RoboDK station: AQIS.rdk

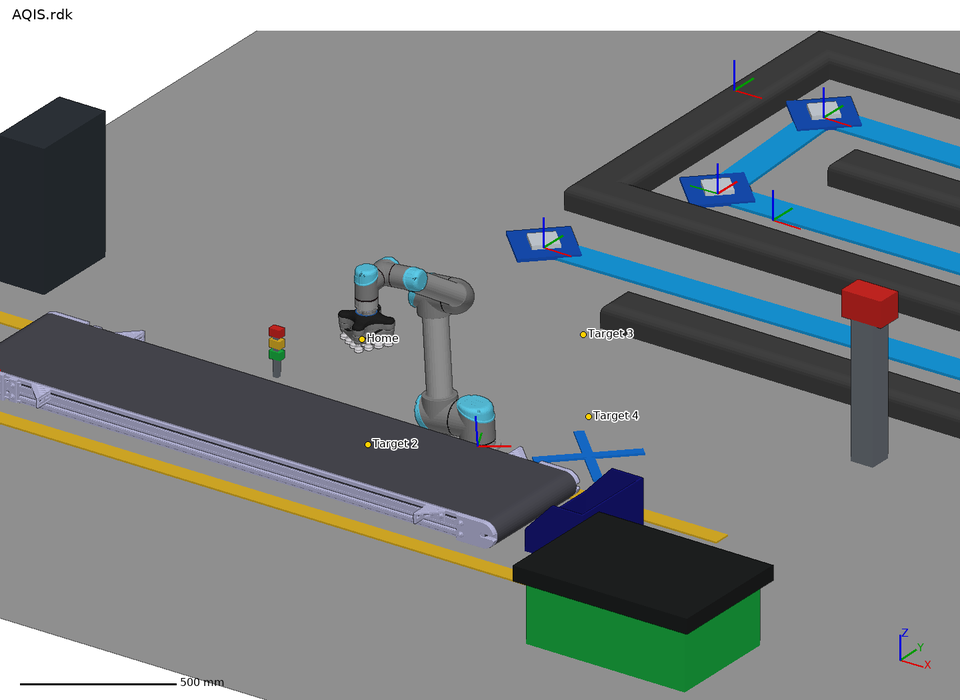
[picture v0: the station drawn from its stored meshes, robots at their saved joint values, targets as dots, program paths as lines]
Station 로봇팔 이동 (saved by RoboDK 5.7.4). Poses are relative to the parent item; angles as X-Y-Z fixed-axis rotations.
Station parameters (name, value as stored): LOAD_READY, 1, RED_DETECTED, 1, AGV_DONE, 1, CONVEYOR_DONE, 1
  - frame MainFrame at (0, 0, 0) mm
    - target Home (Cartesian target) at (651.26, -3006.26, 497.49) mm, rotated rx -179.45 ry 0.15 rz -30.37 deg; joints [-119.255, -87.831, -60.137, -122.512, 86.049, -150.839] of UR5
    - target Target 2 (Cartesian target) at (648.88, -2966.89, 106.48) mm, rotated rx -178.43 ry 0.42 rz -30.32 deg; joints [-119.274, -83.377, -123.993, -64.137, 86.304, -150.836] of UR5
    - target Target 3 (Cartesian target) at (1212.52, -2572.15, 497.3) mm, rotated rx -179.45 ry 0.15 rz -30.37 deg; joints [-13.799, -91.747, -62.441, -119.492, 91.513, -45.448] of UR5
    - target Target 4 (Cartesian target) at (1158.42, -2465.93, 148.85) mm, rotated rx -179.45 ry 0.15 rz -30.37 deg; joints [3.481, -82.996, -122.873, -67.196, 92.538, -28.188] of UR5
    - object path at (2090, -1100, 0) mm, size 3150 x 1417.4 x 86 mm, geometry from path.step
    - object path2 at (1760, -180, 0) mm, rotated rx 0 ry 0 rz 180 deg, size 3150 x 1417.4 x 86 mm, geometry from path.step
    - frame UR5 Base at (820, -2600, 0) mm, rotated rx -1.94 ry -3.6 rz 28.07 deg
      - robot UR5: 6 axes
          modified DH rows (alpha deg, a mm, theta deg, d mm): 0, 0, 0, 89.2; 90, 0, 180, 0; 0, 425, 0, 0; 0, 392, 0, 109.3; -90, 0, 0, 94.75; 90, 0, 180, 82.5
          joint limits [-360, -360, -360, -360, -360, -360] to [360, 360, 360, 360, 360, 360]; home [0, -90, -90, 0, 90, 0]; saved at [-114.958, -89.114, -59.218, -122.443, 86.096, -146.532]
        - tool OnRobot VG10 Vacuum Gripper, TCP at (-36.63, 0, 130.9) mm, size 145.4 x 145.4 x 118.3 mm
    - object Floor at (3000, -3000, 0) mm, size 3000 x 3000 x 0 mm, geometry from Floor (1).sld
    - object Floor at (0, -3000, 0) mm, size 3000 x 3000 x 0 mm, geometry from Floor (1).sld
    - object Floor at (0, 0, 0) mm, size 3000 x 3000 x 0 mm, geometry from Floor (1).sld
    - object Bin Red at (3820, 150, 0) mm, rotated rx 0 ry 0 rz -180 deg, size 225 x 337.5 x 191.2 mm, geometry from Bin-Red.sld
    - object Floor at (3000, 0, 0) mm, size 3000 x 3000 x 0 mm, geometry from Floor (1).sld
    - object Bin Blue at (1380, -2800, 0) mm, rotated rx 0 ry 0 rz -180 deg, size 225 x 337.5 x 191.2 mm, geometry from Bin-Blue.sld
    - frame Conveyor Belt (2m) Base at (-740, -3190, 100) mm
      - robot Conveyor Belt (2m): 1 axes
          modified DH rows (alpha deg, a mm, theta deg, d mm): 0, 0, 0, 0 linear
          base shift (0, 0, 0) mm, rotated rx 0 ry 90 rz 0 deg
          joint limits [-500000] to [500000]; home [0]; saved at [0]
    - frame turtlebot Base at (3580, 0, 20) mm
      - object turtlebot3_waffle at (0, 0, 0) mm, size 280.7 x 305.1 x 138.1 mm, geometry from turtlebot3_waffle (1).step
      - object Red at (48.75, 24.69, 122.77) mm, rotated rx -1.02 ry 0.28 rz -130.77 deg, size 139.8 x 166.4 x 15 mm, geometry from canlid_abnormal.step
    - frame nav1 at (160, -1290, 0) mm
    - frame nav2 at (3450, -1240, 0) mm, rotated rx 0 ry 0 rz 90 deg
    - frame nav3 at (3450, -610, 0) mm, rotated rx 0 ry 0 rz 180 deg
    - frame nav4 at (390, -650, 0) mm, rotated rx 0 ry 0 rz 90 deg
    - frame nav5 at (350, 0, 0) mm
    - frame nav6 at (3580, 0, 0) mm
    - object Blue at (1463.1, -2990, -1.25) mm, size 138.1 x 165.7 x 15 mm, geometry from canlid_normal.step
    - object Green at (1465.6, -2990, -1.25) mm, size 138.1 x 165.7 x 15 mm, geometry from canlid_normal.step
    - object Yellow at (1470.6, -2990, -1.25) mm, size 138.1 x 165.7 x 15 mm, geometry from canlid_normal.step
  - Python program Pickplace (listed below)
  - Python program Turtlebot (listed below)
  - Python program Conv (listed below)
  - Python program Main (listed below)
  - object VIS_Conveyor_Zone_Line_Left at (370, -3310, 2) mm, size 3000 x 65 x 9 mm, geometry from VIS_Conveyor_Zone_Line_Left.stl
  - object VIS_Conveyor_Zone_Line_Right at (350, -2710, 2) mm, size 3000 x 65 x 9 mm, geometry from VIS_Conveyor_Zone_Line_Right.stl
  - object VIS_AGV_Route_Line_01 at (1805, -1265, 6) mm, rotated rx 0 ry 0 rz 0.87 deg, size 3290.4 x 115 x 10 mm, geometry from VIS_AGV_Route_Line_01.stl
  - object VIS_AGV_Route_Line_02 at (3450, -925, 6) mm, rotated rx 0 ry 0 rz 90 deg, size 630 x 115 x 10 mm, geometry from VIS_AGV_Route_Line_02.stl
  - object VIS_AGV_Route_Line_03 at (1920, -630, 6) mm, rotated rx 0 ry 0 rz -179.25 deg, size 3060.3 x 115 x 10 mm, geometry from VIS_AGV_Route_Line_03.stl
  - object VIS_AGV_Route_Line_04 at (370, -325, 6) mm, rotated rx 0 ry 0 rz 93.52 deg, size 651.2 x 115 x 10 mm, geometry from VIS_AGV_Route_Line_04.stl
  - object VIS_AGV_Route_Line_05 at (1965, 0, 6) mm, size 3230 x 115 x 10 mm, geometry from VIS_AGV_Route_Line_05.stl
  - object VIS_AGV_Waypoint_01 at (160, -1290, 12) mm, rotated rx 0 ry 0 rz 45 deg, size 210 x 210 x 12 mm, geometry from VIS_AGV_Waypoint_01.stl
  - object VIS_AGV_Waypoint_Core_01 at (160, -1290, 24) mm, rotated rx 0 ry 0 rz 45 deg, size 95 x 95 x 18 mm, geometry from VIS_AGV_Waypoint_Core_01.stl
  - object VIS_AGV_Waypoint_02 at (3450, -1240, 12) mm, rotated rx 0 ry 0 rz 45 deg, size 210 x 210 x 12 mm, geometry from VIS_AGV_Waypoint_02.stl
  - object VIS_AGV_Waypoint_Core_02 at (3450, -1240, 24) mm, rotated rx 0 ry 0 rz 45 deg, size 95 x 95 x 18 mm, geometry from VIS_AGV_Waypoint_Core_02.stl
  - object VIS_AGV_Waypoint_03 at (3450, -610, 12) mm, rotated rx 0 ry 0 rz 45 deg, size 210 x 210 x 12 mm, geometry from VIS_AGV_Waypoint_03.stl
  - object VIS_AGV_Waypoint_Core_03 at (3450, -610, 24) mm, rotated rx 0 ry 0 rz 45 deg, size 95 x 95 x 18 mm, geometry from VIS_AGV_Waypoint_Core_03.stl
  - object VIS_AGV_Waypoint_04 at (390, -650, 12) mm, rotated rx 0 ry 0 rz 45 deg, size 210 x 210 x 12 mm, geometry from VIS_AGV_Waypoint_04.stl
  - object VIS_AGV_Waypoint_Core_04 at (390, -650, 24) mm, rotated rx 0 ry 0 rz 45 deg, size 95 x 95 x 18 mm, geometry from VIS_AGV_Waypoint_Core_04.stl
  - object VIS_AGV_Waypoint_05 at (350, 0, 12) mm, rotated rx 0 ry 0 rz 45 deg, size 210 x 210 x 12 mm, geometry from VIS_AGV_Waypoint_05.stl
  - object VIS_AGV_Waypoint_Core_05 at (350, 0, 24) mm, rotated rx 0 ry 0 rz 45 deg, size 95 x 95 x 18 mm, geometry from VIS_AGV_Waypoint_Core_05.stl
  - object VIS_AGV_Waypoint_06 at (3580, 0, 12) mm, rotated rx 0 ry 0 rz 45 deg, size 210 x 210 x 12 mm, geometry from VIS_AGV_Waypoint_06.stl
  - object VIS_AGV_Waypoint_Core_06 at (3580, 0, 24) mm, rotated rx 0 ry 0 rz 45 deg, size 95 x 95 x 18 mm, geometry from VIS_AGV_Waypoint_Core_06.stl
  - object VIS_AGV_Pickup_Pad_Target4 at (1158.4, -2465.9, 7) mm, rotated rx 0 ry 0 rz -45 deg, size 360 x 34 x 8 mm, geometry from VIS_AGV_Pickup_Pad_Target4.stl
  - object VIS_AGV_Pickup_Pad_Target4_Cross at (1158.4, -2465.9, 8) mm, rotated rx 0 ry 0 rz -45 deg, size 34 x 360 x 8 mm, geometry from VIS_AGV_Pickup_Pad_Target4_Cross.stl
  - object VIS_AGV_Dock_Pad_Nav6 at (3580, 0, 7) mm, size 420 x 42 x 8 mm, geometry from VIS_AGV_Dock_Pad_Nav6.stl
  - object VIS_AGV_Dock_Pad_Nav6_Cross at (3580, 0, 8) mm, size 42 x 420 x 8 mm, geometry from VIS_AGV_Dock_Pad_Nav6_Cross.stl
  - object VIS_Defect_Dropoff_Arrow at (3580, 295, 18) mm, rotated rx 0 ry 0 rz 90 deg, size 270 x 120 x 14 mm, geometry from VIS_Defect_Dropoff_Arrow.stl
  - object VIS_EStop_Button_Post at (1900, -1960, 260) mm, size 85 x 85 x 520 mm, geometry from VIS_EStop_Button_Post.stl
  - object VIS_EStop_Button_Red at (1900, -1960, 555) mm, size 155 x 95 x 95 mm, geometry from VIS_EStop_Button_Red.stl
  - object VIS_Defect_Storage_Floor at (3580, 735, 7) mm, size 1180 x 920 x 14 mm, geometry from VIS_Defect_Storage_Floor.stl
  - object VIS_Defect_Bin_Base at (3580, 735, 130) mm, size 780 x 520 x 260 mm, geometry from VIS_Defect_Bin_Base.stl
  - object VIS_Defect_Bin_Rim at (3580, 735, 300) mm, size 850 x 590 x 60 mm, geometry from VIS_Defect_Bin_Rim.stl
  - object VIS_Defect_Warning_Panel at (3580, 1190, 340) mm, size 520 x 45 x 300 mm, geometry from VIS_Defect_Warning_Panel.stl
  - object VIS_Normal_Bin_Base at (2080, -3480, 110) mm, size 620 x 420 x 220 mm, geometry from VIS_Normal_Bin_Base.stl
  - object VIS_Normal_Bin_Rim at (2080, -3480, 255) mm, size 680 x 480 x 55 mm, geometry from VIS_Normal_Bin_Rim.stl
  - object VIS_Control_Cabinet at (-1040, -2320, 260) mm, size 180 x 340 x 520 mm, geometry from VIS_Control_Cabinet.stl
  - object VIS_Control_Cabinet_Screen at (-1145, -2320, 350) mm, size 24 x 210 x 125 mm, geometry from VIS_Control_Cabinet_Screen.stl
  - object VIS_Control_Cabinet_Button_Red at (-1160, -2390, 205) mm, size 28 x 45 x 45 mm, geometry from VIS_Control_Cabinet_Button_Red.stl
  - object VIS_Control_Cabinet_Button_Green at (-1160, -2315, 205) mm, size 28 x 45 x 45 mm, geometry from VIS_Control_Cabinet_Button_Green.stl
  - object VIS_AQIS_Sign_Board at (1530, 910, 640) mm, size 1450 x 90 x 520 mm, geometry from VIS_AQIS_Sign_Board.stl
  - object VIS_AQIS_Sign_Base at (1530, 910, 330) mm, size 1700 x 100 x 60 mm, geometry from VIS_AQIS_Sign_Base.stl
  - object VIS_Sign_Letter_A_Top at (1155, 828, 820) mm, size 210 x 35 x 34 mm, geometry from VIS_Sign_Letter_A_Top.stl
  - object VIS_Sign_Letter_A_Mid at (1155, 828, 682) mm, size 210 x 35 x 34 mm, geometry from VIS_Sign_Letter_A_Mid.stl
  - object VIS_Sign_Letter_A_Left at (1050, 828, 670) mm, size 34 x 35 x 300 mm, geometry from VIS_Sign_Letter_A_Left.stl
  - object VIS_Sign_Letter_A_Right at (1260, 828, 670) mm, size 34 x 35 x 300 mm, geometry from VIS_Sign_Letter_A_Right.stl
  - object VIS_Sign_Letter_Q_Top at (1430, 828, 820) mm, size 210 x 35 x 34 mm, geometry from VIS_Sign_Letter_Q_Top.stl
  - object VIS_Sign_Letter_Q_Bottom at (1430, 828, 520) mm, size 210 x 35 x 34 mm, geometry from VIS_Sign_Letter_Q_Bottom.stl
  - object VIS_Sign_Letter_Q_Left at (1325, 828, 670) mm, size 34 x 35 x 300 mm, geometry from VIS_Sign_Letter_Q_Left.stl
  - object VIS_Sign_Letter_Q_Right at (1535, 828, 670) mm, size 34 x 35 x 300 mm, geometry from VIS_Sign_Letter_Q_Right.stl
  - object VIS_Sign_Letter_Q_Tail at (1488.8, 828, 555) mm, size 90 x 35 x 34 mm, geometry from VIS_Sign_Letter_Q_Tail.stl
  - object VIS_Sign_Letter_I_Top at (1705, 828, 820) mm, size 210 x 35 x 34 mm, geometry from VIS_Sign_Letter_I_Top.stl
  - object VIS_Sign_Letter_I_Bottom at (1705, 828, 520) mm, size 210 x 35 x 34 mm, geometry from VIS_Sign_Letter_I_Bottom.stl
  - object VIS_Sign_Letter_I_Center at (1705, 828, 670) mm, size 34 x 35 x 300 mm, geometry from VIS_Sign_Letter_I_Center.stl
  - object VIS_Sign_Letter_S_Top at (1980, 828, 820) mm, size 210 x 35 x 34 mm, geometry from VIS_Sign_Letter_S_Top.stl
  - object VIS_Sign_Letter_S_Mid at (1980, 828, 676) mm, size 210 x 35 x 34 mm, geometry from VIS_Sign_Letter_S_Mid.stl
  - object VIS_Sign_Letter_S_Bottom at (1980, 828, 520) mm, size 210 x 35 x 34 mm, geometry from VIS_Sign_Letter_S_Bottom.stl
  - object VIS_Sign_Letter_S_Left at (1875, 828, 748) mm, size 34 x 35 x 144 mm, geometry from VIS_Sign_Letter_S_Left.stl
  - object VIS_Sign_Letter_S_Right at (2085, 828, 592) mm, size 34 x 35 x 144 mm, geometry from VIS_Sign_Letter_S_Right.stl
  - frame Frame 11 at (200, -70, -380) mm
    - object VIS_Status_Light_Pole at (-200, -2480, 450) mm, size 18 x 18 x 150 mm, geometry from VIS_Status_Light_Pole.stl
    - object VIS_Status_Light_Red at (-200, -2480, 540) mm, size 42 x 30 x 28 mm, geometry from VIS_Status_Light_Red.stl
    - object VIS_Status_Light_Yellow at (-200, -2480, 500) mm, size 42 x 30 x 28 mm, geometry from VIS_Status_Light_Yellow.stl
    - object VIS_Status_Light_Green at (-200, -2480, 460) mm, size 42 x 30 x 28 mm, geometry from VIS_Status_Light_Green.stl

--- Python program Pickplace ---
from robodk import robolink
import time

RDK = robolink.Robolink()

# =========================
# RoboDK 아이템 찾기
# =========================
robot = RDK.Item("UR5")
tool = RDK.Item("OnRobot VG10 Vacuum Gripper")
red_box = RDK.Item("Red")
turtle_base = RDK.Item("turtlebot Base")

home = RDK.Item("Home")
target2 = RDK.Item("Target 2")   # Pick 위치
target3 = RDK.Item("Target 3")   # 이동 중간 위치
target4 = RDK.Item("Target 4")   # Place 위치

def check(item, name):
    if not item.Valid():
        raise Exception(f"'{name}' 을 찾을 수 없습니다. 왼쪽 트리 이름을 확인하세요.")

check(robot, "UR5")
check(tool, "OnRobot VG10 Vacuum Gripper")
check(red_box, "Red")
check(turtle_base, "turtlebot Base")
check(home, "Home")
check(target2, "Target 2")
check(target3, "Target 3")
check(target4, "Target 4")

# 속도 조절
robot.setSpeed(100)

# =========================
# Pick & Place 동작
# =========================

print("1. Home 이동")
robot.MoveJ(home)

print("2. Pick 위치 Target 2 이동")
robot.MoveJ(target2)
time.sleep(0.5)

print("3. Red 흡착")
red_abs = red_box.PoseAbs()
red_box.setParentStatic(tool)
red_box.setPoseAbs(red_abs)
time.sleep(0.5)

print("4. Target 3 이동")
robot.MoveJ(target3)

print("5. Place 위치 Target 4 이동")
robot.MoveJ(target4)
time.sleep(0.5)

print("6. Red를 터틀봇 위에 놓기")
red_abs = red_box.PoseAbs()
red_box.setParentStatic(turtle_base)
red_box.setPoseAbs(red_abs)
time.sleep(0.5)

print("7. Target 3 복귀")
robot.MoveJ(target3)

print("8. Home 복귀")
robot.MoveJ(home)

# 터틀봇 출발 신호
RDK.setParam("LOAD_READY", "1")

print("Pick & Place 완료")

--- Python program Turtlebot ---
from robodk import robolink
from robodk.robomath import *
import time
import math

RDK = robolink.Robolink()

# =========================
# RoboDK 아이템 이름
# =========================
turtle_base = RDK.Item("turtlebot Base")
red_box = RDK.Item("Red")

if not turtle_base.Valid():
    raise Exception("turtlebot Base를 찾을 수 없습니다. 이름을 확인하세요.")

# =========================
# 시작 위치 + 경유지 좌표
# [X, Y, Z]
# =========================
START = [1210, -2510, 20]

WAYPOINTS = [
    [2560, -1140, 20],   # Frame 5
    [-340, -780, 20],    # Frame 4
    [330, -380, 20],     # Frame 3
    [1960, -450, 20],    # Frame 2
    [2640, -20, 20],     # Frame 1
]

# =========================
# Red 박스를 터틀봇에 붙이기
# =========================
if red_box.Valid():
    red_abs_pose = red_box.PoseAbs()
    red_box.setParentStatic(turtle_base)
    red_box.setPoseAbs(red_abs_pose)
    print("Red 박스를 turtlebot Base에 붙였습니다.")
else:
    print("Red 박스를 찾지 못했습니다. 박스 없이 이동합니다.")

# =========================
# pose 생성 함수
# =========================
def make_pose(x, y, z, yaw_deg=0):
    """
    x, y, z 위치와 z축 회전각으로 RoboDK pose 생성
    yaw_deg: 터틀봇 방향 각도
    """
    return transl(x, y, z) * rotz(math.radians(yaw_deg))

# =========================
# 두 점 사이 방향각 계산
# =========================
def calc_yaw_deg(p1, p2):
    dx = p2[0] - p1[0]
    dy = p2[1] - p1[1]
    return math.degrees(math.atan2(dy, dx))

# =========================
# 부드러운 이동 함수
# =========================
def move_smooth(item, target_pose, speed=350, dt=0.03):
    start_pose = item.PoseAbs()

    start = Pose_2_TxyzRxyz(start_pose)
    target = Pose_2_TxyzRxyz(target_pose)

    dx = target[0] - start[0]
    dy = target[1] - start[1]
    dist = math.sqrt(dx * dx + dy * dy)

    steps = max(1, int(dist / (speed * dt)))

    for i in range(1, steps + 1):
        ratio = i / steps

        now = [
            start[j] + (target[j] - start[j]) * ratio
            for j in range(6)
        ]

        item.setPoseAbs(TxyzRxyz_2_Pose(now))
        RDK.Render()
        time.sleep(dt)

# =========================
# 실행
# =========================

# 1. 시작 위치로 세팅
start_yaw = calc_yaw_deg(START, WAYPOINTS[0])
turtle_base.setPoseAbs(make_pose(START[0], START[1], START[2], start_yaw))
RDK.Render()
time.sleep(0.5)

print("TurtleBot 이동 시작")

# 2. 경유지 순서대로 이동
current = START

for idx, wp in enumerate(WAYPOINTS):
    yaw = calc_yaw_deg(current, wp)
    target_pose = make_pose(wp[0], wp[1], wp[2], 0)

    print(f"Moving to Frame {5 - idx}: X={wp[0]}, Y={wp[1]}, Z={wp[2]}, Yaw={yaw:.1f}")
    move_smooth(turtle_base, target_pose, speed=350)

    current = wp

print("TurtleBot 이동 완료")

--- Python program Conv ---
from robodk import robolink
from robodk.robomath import *
import time

RDK = robolink.Robolink()

# =========================
# 이름 설정
# =========================
CONV_BASE_NAME = "Conveyor Belt (2m) Base"
MAIN_FRAME_NAME = "MainFrame"

BOX_NAMES = ["Yellow", "Red", "Green", "Blue"]

conv_base = RDK.Item(CONV_BASE_NAME)
main_frame = RDK.Item(MAIN_FRAME_NAME)

if not conv_base.Valid():
    raise Exception("Conveyor Belt (2m) Base를 찾을 수 없습니다.")

if not main_frame.Valid():
    raise Exception("MainFrame을 찾을 수 없습니다. 왼쪽 트리 이름을 확인하세요.")

boxes = {}

for name in BOX_NAMES:
    box = RDK.Item(name)
    if not box.Valid():
        raise Exception(f"{name} 박스를 찾을 수 없습니다.")
    boxes[name] = box


# =========================
# 초기 위치
# 현재 화면 기준 예상값
# 필요하면 여기 숫자만 수정하면 됨
# [X, Y, Z, RX, RY, RZ]
# =========================
INITIAL_POSES = {
    "Yellow": [200, 200, 0, 0, 0, 0],
    "Red":    [400, 200, 0, 0, 0, 0],
    "Green":  [600, 200, 0, 0, 0, 0],
    "Blue":   [800, 200, 0, 0, 0, 0],
}

# =========================
# 컨베이어 설정
# =========================
STEP_X = 200          # 한 번에 200mm 이동
SUB_STEP = 10         # 10mm씩 나눠서 부드럽게 이동
MOVE_DELAY = 0.02
STOP_DELAY = 0.4

PICK_X = 1000         # 나중에 로봇팔 Pick 위치
BELT_END_X = 2000     # 벨트 끝
RELEASE_X = 2200      # 벨트 끝보다 조금 더 나가면 떨어짐

FALL_DEPTH = 100      # 떨어지는 깊이
GRAVITY = 2500        # 낙하 가속도 느낌, mm/s^2
FALL_DT = 0.03


# =========================
# 유틸 함수
# =========================
def set_box_parent_to_conveyor(box):
    abs_pose = box.PoseAbs()
    box.setParentStatic(conv_base)
    box.setPoseAbs(abs_pose)


def reset_boxes():
    for name, box in boxes.items():
        box.setVisible(True)

        # 다시 컨베이어 기준으로 종속
        set_box_parent_to_conveyor(box)

        # 컨베이어 기준 초기 위치로 세팅
        box.setPose(TxyzRxyz_2_Pose(INITIAL_POSES[name]))

    RDK.Render()
    print("박스 초기 위치 세팅 완료")


def get_local_xyz(box):
    return Pose_2_TxyzRxyz(box.Pose())


def set_local_xyz(box, xyzrxyz):
    box.setPose(TxyzRxyz_2_Pose(xyzrxyz))


def get_local_x(box):
    return get_local_xyz(box)[0]


def move_box_local_x(box, dx):
    xyz = get_local_xyz(box)
    xyz[0] += dx
    set_local_xyz(box, xyz)


def move_conveyor_200(active_names):
    """
    컨베이어를 200mm 이동.
    실제로는 박스들을 10mm씩 나눠 이동시켜서 부드럽게 보이게 함.
    """
    count = int(abs(STEP_X) / SUB_STEP)
    dx = SUB_STEP if STEP_X > 0 else -SUB_STEP

    for _ in range(count):
        for name in active_names:
            move_box_local_x(boxes[name], dx)

        RDK.Render()
        time.sleep(MOVE_DELAY)


def detach_and_fall(name):
    """
    컨베이어 끝을 지난 박스를 MainFrame 기준으로 바꾸고,
    Z값을 점점 낮춰서 중력처럼 떨어지는 연출.
    """
    box = boxes[name]

    print(f"{name}: 컨베이어 종속 해제 후 낙하 시작")

    # 현재 절대 위치 저장
    abs_pose = box.PoseAbs()

    # 컨베이어에서 분리해서 MainFrame 아래로 이동
    box.setParentStatic(main_frame)
    box.setPoseAbs(abs_pose)

    # 절대좌표 기준으로 떨어뜨리기
    xyz = Pose_2_TxyzRxyz(box.PoseAbs())
    start_z = xyz[2]

    velocity = 0.0

    while xyz[2] > start_z - FALL_DEPTH:
        velocity += GRAVITY * FALL_DT
        xyz[2] -= velocity * FALL_DT

        # 벨트에서 튀어나가는 느낌을 조금 주고 싶으면 X도 살짝 이동
        xyz[0] += 30 * FALL_DT

        box.setPoseAbs(TxyzRxyz_2_Pose(xyz))

        RDK.Render()
        time.sleep(FALL_DT)

    print(f"{name}: 낙하 완료")


# =========================
# 실행
# =========================
reset_boxes()

active_names = BOX_NAMES[:]
cycle = 0

print("컨베이어 이동 시작")

while len(active_names) > 0:
    cycle += 1

    print(f"\nCycle {cycle}: 컨베이어 200mm 이동")
    move_conveyor_200(active_names)

    print("컨베이어 정지")
    time.sleep(STOP_DELAY)

    # 나중에 로봇팔 넣을 때 확인용
    for name in active_names:
        x = get_local_x(boxes[name])
        if abs(x - PICK_X) <= 20:
            print(f"{name}이 Pick 위치 X={PICK_X} 근처에 있음")

    # 벨트 끝보다 조금 더 나간 박스는 떨어뜨림
    arrived = []

    for name in active_names:
        x = get_local_x(boxes[name])

        if x >= RELEASE_X:
            arrived.append(name)

    for name in arrived:
        active_names.remove(name)
        detach_and_fall(name)

    if cycle > 30:
        print("안전 종료: cycle이 너무 많습니다. STEP_X 방향을 확인하세요.")
        break

print("\n컨베이어 테스트 완료")

--- Python program Main ---
from robodk import robolink
from robodk.robomath import *
import time
import math
import threading
import json
import uuid
from urllib import request, error

RDK = robolink.Robolink()
SCRIPT_ID = f"robodk-{uuid.uuid4().hex}"

# =========================================================
# Web UI / FastAPI 연동 설정
# =========================================================
# FastAPI 서버를 WSL 또는 Windows에서 실행한 뒤 주소를 맞추면 됨.
# 보통 같은 PC에서 실행하면 http://localhost:8000 사용.
API_BASE = "http://localhost:8000"
API_TIMEOUT = 0.3
ENABLE_WEB_UI_SYNC = True
COMMAND_POLL_DT = 0.25
RENDER_MIN_DT = 0.08
WEB_STATUS_MIN_DT = 0.5

# =========================================================
# RoboDK 아이템 이름
# =========================================================
ROBOT_NAME = "UR5"
TOOL_NAME = "OnRobot VG10 Vacuum Gripper"

CONV_BASE_NAME = "Conveyor Belt (2m) Base"
MAIN_FRAME_NAME = "MainFrame"

TURTLE_NAME = "turtlebot Base"

BOX_NAMES = ["Yellow", "Red", "Green", "Blue"]

TARGET_HOME = "Home"
TARGET_PICK = "Target 2"      # Red 감지 후 집는 위치
TARGET_MID = "Target 3"       # 로봇 중간 경유 위치
TARGET_PLACE = "Target 4"     # TurtleBot 위에 놓는 위치

# =========================================================
# 공정 파라미터
# =========================================================
# Red를 detect해서 컨베이어를 멈출 X 좌표
DETECT_X = 1400
DETECT_TOL = 10

# 컨베이어 연속 이동 속도 설정
CONVEYOR_SPEED = 250      # mm/s
CONVEYOR_DT = 0.03        # sec
CONVEYOR_DX = CONVEYOR_SPEED * CONVEYOR_DT

# 컨베이어 끝 / 낙하 설정
RELEASE_X = 2200
FALL_DEPTH = 100
GRAVITY = 2500
FALL_DT = 0.03

# 로봇 속도
ROBOT_SPEED = 100

# TurtleBot 이동 속도
AGV_SPEED = 2350
AGV_DT = 0.005

# =========================================================
# 초기 박스 위치: 컨베이어 기준 local pose [X, Y, Z, RX, RY, RZ]
# =========================================================
INITIAL_POSES = {
    "Yellow": [200, 200, 0, 0, 0, 0],
    "Red":    [400, 200, 0, 0, 0, 0],
    "Green":  [600, 200, 0, 0, 0, 0],
    "Blue":   [800, 200, 0, 0, 0, 0],
}

# =========================================================
# TurtleBot 시작 위치 + 불량 저장 위치 경로 [X, Y, Z]
# =========================================================
AGV_START = [1210, -2510, 20]

# Station에 찍어둔 nav 프레임을 TurtleBot 이동 waypoint의 기준으로 사용한다.
# RoboDK에서 nav1~nav6를 옮기면 스크립트가 그 좌표를 읽어 이동 경로에 반영한다.
DEFECT_STORAGE_NAV_NAMES = ["nav1", "nav2", "nav3", "nav4", "nav5", "nav6"]

# nav 프레임이 없는 환경에서만 쓰는 fallback 좌표 [X, Y, Z].
# 마지막 좌표를 불량 저장 위치로 사용한다.
DEFECT_STORAGE_PATH = [
    [160, -1290, 20],    # nav1
    [3450, -1240, 20],   # nav2
    [3450, -610, 20],    # nav3
    [390, -650, 20],     # nav4
    [350, 0, 20],        # nav5
    [3580, 0, 20],       # nav6 / 불량 저장 위치
]

# =========================================================
# RoboDK 아이템 찾기
# =========================================================
robot = RDK.Item(ROBOT_NAME)
tool = RDK.Item(TOOL_NAME)

conv_base = RDK.Item(CONV_BASE_NAME)
main_frame = RDK.Item(MAIN_FRAME_NAME)

turtle_base = RDK.Item(TURTLE_NAME)

home = RDK.Item(TARGET_HOME)
target_pick = RDK.Item(TARGET_PICK)
target_mid = RDK.Item(TARGET_MID)
target_place = RDK.Item(TARGET_PLACE)

boxes = {}
for name in BOX_NAMES:
    boxes[name] = RDK.Item(name)

red_box = boxes["Red"]

# 병렬 실행 시 RoboDK API 충돌 방지용 Lock
RDK_LOCK = threading.RLock()
LAST_RENDER_AT = 0.0
LAST_STATUS_SENT_AT = 0.0
LAST_STATUS_PAYLOAD = None

# 같은 Python 스크립트 안의 공정 분기에는 RoboDK Param보다 로컬 상태를 우선 사용.
# 일부 RoboDK 실행 환경에서 RDK.setParam("KEY", "1") 후 RDK.getParam("KEY")가
# 바로 문자열 "1"로 돌아오지 않아 분기 오류가 생길 수 있다.
STATE = {
    "red_detected": False,
    "load_ready": False,
    "agv_done": False,
    "conveyor_done": False,
    "paused": False,
    "stop_requested": False,
    "reset_requested": False,
    "last_command": None,
}
DETECTED_NAMES = set()

# =========================================================
# Web UI 연동 유틸
# =========================================================
class StopRequested(Exception):
    pass


class ResetRequested(Exception):
    pass


def api_request(method, path, payload=None, log_fail=True):
    """FastAPI 서버와 통신한다. 실패해도 RoboDK 시뮬레이션 자체는 계속 실행한다."""
    if not ENABLE_WEB_UI_SYNC:
        return None

    url = API_BASE + path
    data = None
    headers = {}

    if payload is not None:
        data = json.dumps(payload).encode("utf-8")
        headers["Content-Type"] = "application/json"

    try:
        req = request.Request(url, data=data, headers=headers, method=method)
        with request.urlopen(req, timeout=API_TIMEOUT) as res:
            raw = res.read().decode("utf-8")
            if raw:
                return json.loads(raw)
            return None
    except Exception as exc:
        if log_fail:
            print(f"[WEB_UI] {method} 실패: {path} / {exc}")
        return None


def api_post(path, payload=None):
    return api_request("POST", path, payload)


def api_get(path, log_fail=True):
    return api_request("GET", path, None, log_fail=log_fail)


def notify_web_status(stage, message="", running=True, red_x=None, force=False):
    global LAST_STATUS_PAYLOAD, LAST_STATUS_SENT_AT

    payload = {
        "script_id": SCRIPT_ID,
        "connected": True,
        "running": running,
        "stage": stage,
        "message": message,
    }
    if red_x is not None:
        payload["red_x"] = red_x

    now = time.monotonic()
    with RDK_LOCK:
        if (
            not force
            and payload == LAST_STATUS_PAYLOAD
            and now - LAST_STATUS_SENT_AT < WEB_STATUS_MIN_DT
        ):
            return
        LAST_STATUS_PAYLOAD = payload.copy()
        LAST_STATUS_SENT_AT = now

    api_post("/api/robodk/status", payload)


def notify_web_reset():
    print("[WEB_UI] RoboDK Reset 상태 전송")
    notify_web_status("RESET", "RoboDK scene reset", running=False, force=True)


def notify_web_detection(color_name, x, result):
    color = color_name.lower()
    is_defect = result == "defect"
    print(f"[WEB_UI] Detection 이벤트 전송: {color} / {result} / X={x:.1f}")
    api_post(
        "/api/sim/detection",
        {
            "part_id": f"robodk_{color}_{int(time.time() * 1000)}",
            "color": color,
            "result": result,
            "source": "robodk",
            "script_id": SCRIPT_ID,
            "confidence": 0.99 if is_defect else 0.96,
            "x": x,
        },
    )


def mark_detected_once(name):
    with RDK_LOCK:
        if name in DETECTED_NAMES:
            return False
        DETECTED_NAMES.add(name)
        return True


def notify_web_agv_dispatch():
    print("[WEB_UI] AGV Dispatch 이벤트 전송")
    api_post("/api/sim/agv/dispatch", {"source": "robodk", "script_id": SCRIPT_ID})


def notify_web_agv_state(status, message="", waypoint_index=None, waypoint_total=None, position=None):
    payload = {
        "source": "robodk",
        "script_id": SCRIPT_ID,
        "status": status,
        "message": message,
    }
    if waypoint_index is not None:
        payload["waypoint_index"] = waypoint_index
    if waypoint_total is not None:
        payload["waypoint_total"] = waypoint_total
    if position is not None:
        payload["x"] = position[0]
        payload["y"] = position[1]
        payload["z"] = position[2]
    api_post("/api/sim/agv/state", payload)


def notify_web_stop():
    print("[WEB_UI] RoboDK Stop 상태 전송")
    notify_web_status("STOPPED", "RoboDK sequence stopped", running=False, force=True)


def apply_command(command):
    if not command:
        return
    with RDK_LOCK:
        STATE["last_command"] = command
        if command == "PAUSE":
            STATE["paused"] = True
        elif command == "START":
            STATE["paused"] = False
        elif command == "STOP":
            STATE["paused"] = False
            STATE["stop_requested"] = True
        elif command == "RESET":
            STATE["paused"] = False
            STATE["reset_requested"] = True
        elif command == "DISPATCH_AGV":
            # 실제 AGV 이동은 Red 적재 후 Main 시퀀스에서 수행한다. 여기서는 명령 수신만 기록.
            pass
    print(f"[WEB_UI] Command 수신: {command}")


def poll_web_command_once(log_fail=False):
    data = api_get(f"/api/robodk/command?script_id={SCRIPT_ID}", log_fail=log_fail)
    if isinstance(data, dict):
        apply_command(data.get("command"))


def command_listener_worker():
    print("[WEB_UI] Web command listener 시작")
    while True:
        poll_web_command_once(log_fail=False)
        with RDK_LOCK:
            if STATE["stop_requested"] or STATE["reset_requested"]:
                break
        time.sleep(COMMAND_POLL_DT)
    print("[WEB_UI] Web command listener 종료")


def wait_if_paused_or_interrupted():
    while True:
        with RDK_LOCK:
            if STATE["stop_requested"]:
                raise StopRequested()
            if STATE["reset_requested"]:
                raise ResetRequested()
            paused = STATE["paused"]
        if not paused:
            return
        notify_web_status("PAUSED", "RoboDK sequence paused", running=False)
        time.sleep(COMMAND_POLL_DT)


def controlled_sleep(seconds):
    end_time = time.time() + seconds
    while time.time() < end_time:
        wait_if_paused_or_interrupted()
        time.sleep(min(COMMAND_POLL_DT, max(0, end_time - time.time())))


def wait_for_web_start_command():
    print("[WEB_UI] Web UI에서 Simulation Start를 누를 때까지 대기합니다.")
    notify_web_status("READY", "Waiting for Web UI START", running=False, force=True)
    while True:
        poll_web_command_once(log_fail=True)
        with RDK_LOCK:
            command = STATE["last_command"]
            if command == "START":
                STATE["last_command"] = None
                STATE["stop_requested"] = False
                STATE["reset_requested"] = False
                STATE["paused"] = False
                return
        time.sleep(COMMAND_POLL_DT)

# =========================================================
# 검증 함수
# =========================================================
def check(item, name):
    if not item.Valid():
        raise Exception(f"'{name}' 을 찾을 수 없습니다. RoboDK 왼쪽 트리 이름을 확인하세요.")


def check_all_items():
    check(robot, ROBOT_NAME)
    check(tool, TOOL_NAME)
    check(conv_base, CONV_BASE_NAME)
    check(main_frame, MAIN_FRAME_NAME)
    check(turtle_base, TURTLE_NAME)
    check(home, TARGET_HOME)
    check(target_pick, TARGET_PICK)
    check(target_mid, TARGET_MID)
    check(target_place, TARGET_PLACE)

    for name, box in boxes.items():
        check(box, name)

# =========================================================
# Pose / 좌표 유틸
# =========================================================
def make_pose(x, y, z, yaw_deg=0):
    return transl(x, y, z) * rotz(math.radians(yaw_deg))


def calc_yaw_deg(p1, p2):
    dx = p2[0] - p1[0]
    dy = p2[1] - p1[1]
    return math.degrees(math.atan2(dy, dx))


def get_defect_storage_path():
    """RoboDK Station의 nav1~nav6 프레임을 TurtleBot waypoint로 읽는다.

    nav 프레임은 시각 경로(path/path2) 위에 사용자가 직접 찍어둔 좌표이므로
    스크립트의 하드코딩보다 우선한다. 프레임이 하나라도 없으면 fallback
    DEFECT_STORAGE_PATH를 사용한다.
    """
    waypoints = []
    for name in DEFECT_STORAGE_NAV_NAMES:
        nav = RDK.Item(name)
        if not nav.Valid():
            print(f"[AGV] {name} 프레임이 없어 fallback DEFECT_STORAGE_PATH를 사용합니다.")
            return [wp[:] for wp in DEFECT_STORAGE_PATH]
        xyz = Pose_2_TxyzRxyz(nav.PoseAbs())
        waypoints.append([xyz[0], xyz[1], AGV_START[2]])
    return waypoints


def get_local_xyz(item):
    with RDK_LOCK:
        return Pose_2_TxyzRxyz(item.Pose())


def get_local_x(item):
    xyz = get_local_xyz(item)
    return xyz[0]


def move_box_local_x(box, dx):
    with RDK_LOCK:
        xyz = Pose_2_TxyzRxyz(box.Pose())
        xyz[0] += dx
        box.setPose(TxyzRxyz_2_Pose(xyz))


def safe_render(force=False):
    global LAST_RENDER_AT

    now = time.monotonic()
    with RDK_LOCK:
        if not force and now - LAST_RENDER_AT < RENDER_MIN_DT:
            return
        RDK.Render()
        LAST_RENDER_AT = now

# =========================================================
# 초기화
# =========================================================
def set_box_parent_to_conveyor(box):
    with RDK_LOCK:
        abs_pose = box.PoseAbs()
        box.setParentStatic(conv_base)
        box.setPoseAbs(abs_pose)


def reset_boxes():
    print("[RESET] 박스 초기 위치 세팅")

    for name, box in boxes.items():
        with RDK_LOCK:
            box.setVisible(True)

        set_box_parent_to_conveyor(box)

        with RDK_LOCK:
            box.setPose(TxyzRxyz_2_Pose(INITIAL_POSES[name]))

    safe_render()
    print("[RESET] 박스 초기 위치 세팅 완료")


def reset_agv():
    print("[RESET] TurtleBot 시작 위치 세팅")

    nav_path = get_defect_storage_path()
    first_waypoint = nav_path[0] if nav_path else DEFECT_STORAGE_PATH[0]
    start_yaw = calc_yaw_deg(AGV_START, first_waypoint)

    with RDK_LOCK:
        turtle_base.setPoseAbs(
            make_pose(AGV_START[0], AGV_START[1], AGV_START[2], start_yaw)
        )

    safe_render()
    print("[RESET] TurtleBot 시작 위치 세팅 완료")


def reset_robot():
    print("[RESET] UR5 Home 이동")

    with RDK_LOCK:
        robot.setSpeed(ROBOT_SPEED)

    wait_if_paused_or_interrupted()
    robot.MoveJ(home)
    print("[RESET] UR5 Home 이동 완료")


def reset_scene():
    print("\n========== 1. Scene Reset ==========")

    notify_web_reset()

    reset_boxes()
    reset_agv()
    reset_robot()

    with RDK_LOCK:
        STATE["red_detected"] = False
        STATE["load_ready"] = False
        STATE["agv_done"] = False
        STATE["conveyor_done"] = False
        STATE["stop_requested"] = False
        STATE["reset_requested"] = False
        DETECTED_NAMES.clear()
        RDK.setParam("RED_DETECTED", "0")
        RDK.setParam("LOAD_READY", "0")
        RDK.setParam("AGV_DONE", "0")
        RDK.setParam("CONVEYOR_DONE", "0")

    controlled_sleep(0.5)

# =========================================================
# 컨베이어 연속 이동: Red가 X=1400에 도달하면 정지
# =========================================================
def conveyor_until_red_detect():
    print("\n========== 2. Conveyor Move Until Red Detect ==========")
    print(f"[CONVEYOR] Detect 기준 X = {DETECT_X} (정상/불량 모두 처리)")
    notify_web_status("CONVEYOR", "Conveyor moving and vision detection active", running=True)

    active_names = BOX_NAMES[:]
    while True:
        wait_if_paused_or_interrupted()
        # 컨베이어 위 활성 박스들을 계속 이동. 200mm 단위 정지가 아니라 연속 이동.
        for name in active_names:
            move_box_local_x(boxes[name], CONVEYOR_DX)

        safe_render()
        controlled_sleep(CONVEYOR_DT)

        for name in active_names:
            x = get_local_x(boxes[name])
            if x >= DETECT_X - DETECT_TOL and mark_detected_once(name):
                if name == "Red":
                    print(f"[DETECT] Red 불량 감지됨. Red X = {x:.1f}")
                    print("[CONVEYOR] Red pick을 위해 컨베이어 정지")

                    with RDK_LOCK:
                        STATE["red_detected"] = True
                        RDK.setParam("RED_DETECTED", "1")

                    notify_web_detection("Red", x, "defect")
                    notify_web_status("RED_DETECTED", "Red defect detected; conveyor stopped for UR5 pick", running=True, red_x=x)
                    print("[CONVEYOR] Red detect 단계 완료")
                    return
                else:
                    print(f"[DETECT] {name} 정상 감지됨. X = {x:.1f}")
                    notify_web_detection(name, x, "normal")

        red_x = get_local_x(red_box)
        if red_x > RELEASE_X:
            raise Exception(
                f"[ERROR] Red가 감지되지 않고 RELEASE_X를 지났습니다. "
                f"현재 Red X={red_x:.1f}, DETECT_X={DETECT_X}"
            )

# =========================================================
# UR5가 Red를 집어서 TurtleBot 위에 적재
# =========================================================
def pick_red_to_turtlebot():
    print("\n========== 3. UR5 Pick Red -> TurtleBot ==========")
    notify_web_status("UR5_PICK", "UR5 picking red defect to TurtleBot", running=True)

    with RDK_LOCK:
        red_detected = STATE["red_detected"]

    if not red_detected:
        raise Exception("[UR5] Red가 detect되지 않았습니다. Pick 동작을 중단합니다.")

    with RDK_LOCK:
        robot.setSpeed(ROBOT_SPEED)

    print("[UR5] Home 이동")
    wait_if_paused_or_interrupted()
    robot.MoveJ(home)

    print("[UR5] Pick 위치 이동")
    wait_if_paused_or_interrupted()
    robot.MoveJ(target_pick)
    controlled_sleep(0.3)

    print("[UR5] Red 흡착")
    with RDK_LOCK:
        red_abs_pose = red_box.PoseAbs()
        red_box.setParentStatic(tool)
        red_box.setPoseAbs(red_abs_pose)

    safe_render()
    controlled_sleep(0.3)

    print("[UR5] 중간 위치 이동")
    wait_if_paused_or_interrupted()
    robot.MoveJ(target_mid)

    print("[UR5] TurtleBot 위 Place 위치 이동")
    wait_if_paused_or_interrupted()
    robot.MoveJ(target_place)
    controlled_sleep(0.3)

    print("[UR5] Red를 TurtleBot 위에 놓기")
    with RDK_LOCK:
        red_abs_pose = red_box.PoseAbs()
        red_box.setParentStatic(turtle_base)
        red_box.setPoseAbs(red_abs_pose)

    safe_render()
    controlled_sleep(0.3)

    print("[UR5] 중간 위치 복귀")
    wait_if_paused_or_interrupted()
    robot.MoveJ(target_mid)

    print("[UR5] Home 복귀")
    wait_if_paused_or_interrupted()
    robot.MoveJ(home)

    with RDK_LOCK:
        STATE["load_ready"] = True
        RDK.setParam("LOAD_READY", "1")

    notify_web_agv_dispatch()
    print("[UR5] Red 적재 완료. LOAD_READY = 1")

# =========================================================
# 박스 낙하 연출
# =========================================================
def detach_and_fall(name):
    box = boxes[name]

    print(f"[CONVEYOR] {name}: 컨베이어 끝 도달. 낙하 시작")

    with RDK_LOCK:
        abs_pose = box.PoseAbs()
        box.setParentStatic(main_frame)
        box.setPoseAbs(abs_pose)

        xyz = Pose_2_TxyzRxyz(box.PoseAbs())
        start_z = xyz[2]

    velocity = 0.0

    while xyz[2] > start_z - FALL_DEPTH:
        velocity += GRAVITY * FALL_DT
        xyz[2] -= velocity * FALL_DT
        xyz[0] += 30 * FALL_DT

        with RDK_LOCK:
            box.setPoseAbs(TxyzRxyz_2_Pose(xyz))

        safe_render()

        controlled_sleep(FALL_DT)

    print(f"[CONVEYOR] {name}: 낙하 완료")

# =========================================================
# 병렬 작업 1: Red 제외 나머지 박스 컨베이어 계속 이동
# =========================================================
def conveyor_rest_worker():
    print("\n========== Parallel A. Conveyor Rest Start ==========")
    notify_web_status("CONVEYOR_REST", "Normal parts continue to conveyor end", running=True)

    active_names = ["Yellow", "Green", "Blue"]

    while len(active_names) > 0:
        for name in active_names:
            move_box_local_x(boxes[name], CONVEYOR_DX)

        safe_render()
        controlled_sleep(CONVEYOR_DT)

        arrived = []

        for name in active_names:
            x = get_local_x(boxes[name])
            if x >= DETECT_X - DETECT_TOL and mark_detected_once(name):
                print(f"[DETECT] {name} 정상 감지됨. X = {x:.1f}")
                notify_web_detection(name, x, "normal")

            if x >= RELEASE_X:
                arrived.append(name)

        for name in arrived:
            active_names.remove(name)
            detach_and_fall(name)

    with RDK_LOCK:
        STATE["conveyor_done"] = True
        RDK.setParam("CONVEYOR_DONE", "1")

    print("[CONVEYOR] 나머지 박스 이동 완료. CONVEYOR_DONE = 1")

# =========================================================
# TurtleBot 부드러운 절대좌표 이동
# =========================================================
def move_smooth_abs(item, target_pose, speed=350, dt=0.03):
    with RDK_LOCK:
        start_pose = item.PoseAbs()

    start = Pose_2_TxyzRxyz(start_pose)
    target = Pose_2_TxyzRxyz(target_pose)

    dx = target[0] - start[0]
    dy = target[1] - start[1]

    dist = math.sqrt(dx * dx + dy * dy)
    steps = max(1, int(dist / (speed * dt)))

    # TurtleBot body 정렬: 이동 구간마다 진행 방향 yaw를 먼저 맞춘 뒤,
    # 위치만 보간한다. 기존처럼 yaw까지 선형 보간하면 코너 진입/이탈 구간에서
    # 몸체가 경로를 비스듬히 물고 지나가 path와 겹쳐 보인다.
    segment_yaw = target[5]
    with RDK_LOCK:
        aligned_start = start[:]
        aligned_start[5] = segment_yaw
        item.setPoseAbs(TxyzRxyz_2_Pose(aligned_start))

    for i in range(1, steps + 1):
        ratio = i / steps

        now = start[:]
        now[0] = start[0] + dx * ratio
        now[1] = start[1] + dy * ratio
        now[2] = start[2] + (target[2] - start[2]) * ratio
        now[3] = target[3]
        now[4] = target[4]
        now[5] = segment_yaw

        with RDK_LOCK:
            item.setPoseAbs(TxyzRxyz_2_Pose(now))

        safe_render()

        controlled_sleep(dt)

    with RDK_LOCK:
        return Pose_2_TxyzRxyz(item.PoseAbs())

# =========================================================
# 병렬 작업 2: TurtleBot이 불량 저장 위치로 이동
# =========================================================
def agv_to_defect_storage_worker():
    print("\n========== Parallel B. TurtleBot To Defect Storage Start ==========")
    notify_web_status("AGV_MOVING", "TurtleBot moving to defect storage", running=True)

    with RDK_LOCK:
        load_ready = STATE["load_ready"]

    if not load_ready:
        print("[AGV] LOAD_READY가 1이 아닙니다. TurtleBot 이동 취소.")
        return

    print("[AGV] Red 적재 확인. 불량 저장 위치로 이동 시작")
    nav_path = get_defect_storage_path()
    waypoint_total = len(nav_path)
    notify_web_agv_state(
        "MOVING_TO_DEFECT_BIN",
        "TurtleBot started moving to defect storage.",
        waypoint_index=0,
        waypoint_total=waypoint_total,
        position=AGV_START,
    )

    current = AGV_START

    for idx, wp in enumerate(nav_path):
        yaw = calc_yaw_deg(current, wp)
        target_pose = make_pose(wp[0], wp[1], wp[2], yaw)

        print(
            f"[AGV] Waypoint {idx + 1} 이동: "
            f"X={wp[0]:.1f}, Y={wp[1]:.1f}, Z={wp[2]:.1f}, Yaw={yaw:.1f}"
        )

        final_pose = move_smooth_abs(turtle_base, target_pose, speed=AGV_SPEED, dt=AGV_DT)
        notify_web_agv_state(
            "MOVING_TO_DEFECT_BIN",
            f"TurtleBot reached waypoint {idx + 1}/{waypoint_total}.",
            waypoint_index=idx + 1,
            waypoint_total=waypoint_total,
            position=final_pose[:3],
        )
        current = wp

    with RDK_LOCK:
        STATE["agv_done"] = True
        RDK.setParam("AGV_DONE", "1")

    final_position = nav_path[-1] if nav_path else DEFECT_STORAGE_PATH[-1]
    notify_web_agv_state(
        "COMPLETED",
        "TurtleBot arrived at defect storage.",
        waypoint_index=waypoint_total,
        waypoint_total=waypoint_total,
        position=final_position,
    )
    print("[AGV] 불량 저장 위치 도착. AGV_DONE = 1")

# =========================================================
# TurtleBot과 컨베이어 병렬 실행
# =========================================================
def run_parallel_agv_and_conveyor():
    print("\n========== 4. Parallel Process Start ==========")
    print("[PARALLEL] TurtleBot 이동과 컨베이어 이동을 동시에 실행합니다.")

    errors = []

    def run_worker(worker):
        try:
            worker()
        except Exception as exc:
            with RDK_LOCK:
                errors.append(exc)
                STATE["stop_requested"] = True

    agv_thread = threading.Thread(target=run_worker, args=(agv_to_defect_storage_worker,), name="AGVThread")
    conveyor_thread = threading.Thread(target=run_worker, args=(conveyor_rest_worker,), name="ConveyorThread")

    agv_thread.start()
    conveyor_thread.start()

    agv_thread.join()
    conveyor_thread.join()

    if errors:
        raise errors[0]

    print("[PARALLEL] TurtleBot 이동과 컨베이어 이동 모두 완료")

# =========================================================
# Main Sequence
# =========================================================
def run_sequence_once():
    reset_scene()

    # 1. 컨베이어가 계속 이동하면서 정상품도 detect 처리하고, Red가 X=1400에서 detect되면 정지
    conveyor_until_red_detect()

    # 2. UR5가 Red를 집어서 TurtleBot 위로 이동
    pick_red_to_turtlebot()

    # 3. Red 적재 후 TurtleBot 이동 + 컨베이어 이동 병렬 실행
    run_parallel_agv_and_conveyor()


def main():
    check_all_items()

    print("\n==============================================")
    print("AQIS RoboDK Main Sequence + Web UI Control/Sync Start")
    print("==============================================")

    while True:
        wait_for_web_start_command()
        listener = threading.Thread(target=command_listener_worker, name="WebCommandThread", daemon=True)
        listener.start()

        try:
            notify_web_status("RUNNING", "RoboDK sequence started by Web UI", running=True)
            run_sequence_once()
            notify_web_status("DONE", "RoboDK sequence completed", running=False)
            print("\n==============================================")
            print("AQIS RoboDK Main Sequence + Web UI Sync Done")
            print("==============================================")
        except ResetRequested:
            print("[WEB_UI] Reset command 처리: 장면 초기화 후 다시 START 대기")
            reset_scene()
            notify_web_status("READY", "Reset done. Waiting for Web UI START", running=False)
        except StopRequested:
            print("[WEB_UI] Stop command 처리: 시퀀스 중지 후 다시 START 대기")
            notify_web_stop()
        finally:
            with RDK_LOCK:
                STATE["stop_requested"] = True
            listener.join(timeout=1.0)
            with RDK_LOCK:
                STATE["stop_requested"] = False
                STATE["reset_requested"] = False
                STATE["paused"] = False
                STATE["last_command"] = None


main()
